FUNCTION_BLOCK FB_Module IMPLEMENTS I_Module
VAR
	_Name : STRING;
	_Counter : udint;
END_VAR

METHOD Accept
VAR_INPUT
	Visitor : I_VisitModules;
END_VAR
Visitor.VisitModules(THIS^);
END_METHOD

PROPERTY CounterValue : UDINT
GET
CounterValue := _Counter;
END_GET
SET
_Counter := CounterValue;
END_SET
END_PROPERTY

METHOD CyclicLogic : BOOL
VAR_INPUT
END_VAR
_Counter := _Counter + 1;
END_METHOD

PROPERTY Name : STRING
GET
Name := _Name;
END_GET
SET
_Name := NAme;
END_SET
END_PROPERTY

END_FUNCTION_BLOCK

(* stored: Version 1.1.0.1, ProductVersion 3.1.4024.12
   POU FB_Module: Id {ca542684-4b12-4224-9ba1-d68d2d2ffb0e}, SpecialFunc None
   Method Accept: Id {ca1dc568-b4a3-47c4-9915-d3f8064fc7cd}
   Property CounterValue: Id {b72f4e84-6612-43a1-ad6e-1f3f1569d818}
   Get Get: Id {d789c8e5-6e1e-41ce-a805-d9e0bb3de30c}
   Set Set: Id {b280cacd-96d8-43fa-876d-495a7a54746d}
   Method CyclicLogic: Id {2d04fa79-ae4b-468c-8baf-4222da60883a}
   Property Name: Id {715e9e0a-8e94-4ff2-beb7-2532b213fcef}
   Get Get: Id {0374513d-08bc-4510-8872-f906a2e8a2c0}
   Set Set: Id {8282942d-e9c6-468b-a4b0-b68911f35941} *)
